(* Logix 5000 project; controller Sucrose_Main Emulate 5570 rev 20.12; software revision 20.01; part 16 of 30 *)
(* tags used below, declared in another part *)
   Alarm_ACK_Master_Timer : TIMER;
   DO_E22_4 : ALIAS FOR FLX_E22:4:O;   // Discrete Output EN2T_FLX 192.168.1.22
   DO_E22_5 : ALIAS FOR FLX_E22:5:O;   // Discrete Output EN2T_FLX 192.168.1.22
   FV230502_AOI : QSI_Flow_Valve;   // FV-23-05-02 PRE FILTER TRAIN 1 INLET LOW POINT DRAIN VALVE
   FV230503_AOI : QSI_Flow_Valve;   // FV-23-05-03 PRE FILTER TRAIN 1 INLET LOW POINT DRAIN VALVE
   FV230504_AOI : QSI_Flow_Valve;   // FV-23-05-04 PRE FILTER TRAIN 1 OUTLET LOW POINT DRAIN VALVE
   FV230505_AOI : QSI_Flow_Valve;   // FV-23-05-05 PRE FILTER TRAIN 1 OUTLET LOW POINT DRAIN VALVE
   FV230509_AOI : QSI_Flow_Valve;   // FV-23-05-09 FINAL FILTER TRAIN 1 INLET LOW POINT DRAIN VALVE
   FV230510_AOI : QSI_Flow_Valve;   // FV-23-05-10 FINAL FILTER TRAIN 1 INLET LOW POINT DRAIN VALVE
   FV230511_AOI : QSI_Flow_Valve;   // FV-23-05-11 FINAL FILTER TRAIN 1 OUTLET LOW POINT DRAIN VALVE
   FV230512_AOI : QSI_Flow_Valve;   // FV-23-05-12 FINAL FILTER TRAIN 1 OUTLET LOW POINT DRAIN VALVE
   Sucrose_MM_Enable : BOOL;
   SucroseCIP_FILTRATION_REMOTE : CIP_REMOTE;
   SucroseFiltration : Area_Program;
(* FiltrationArea_EN2T_IO_Discrete_DO_E22_4, continued *)

ROUTINE _07_FV230502   (* ladder *)
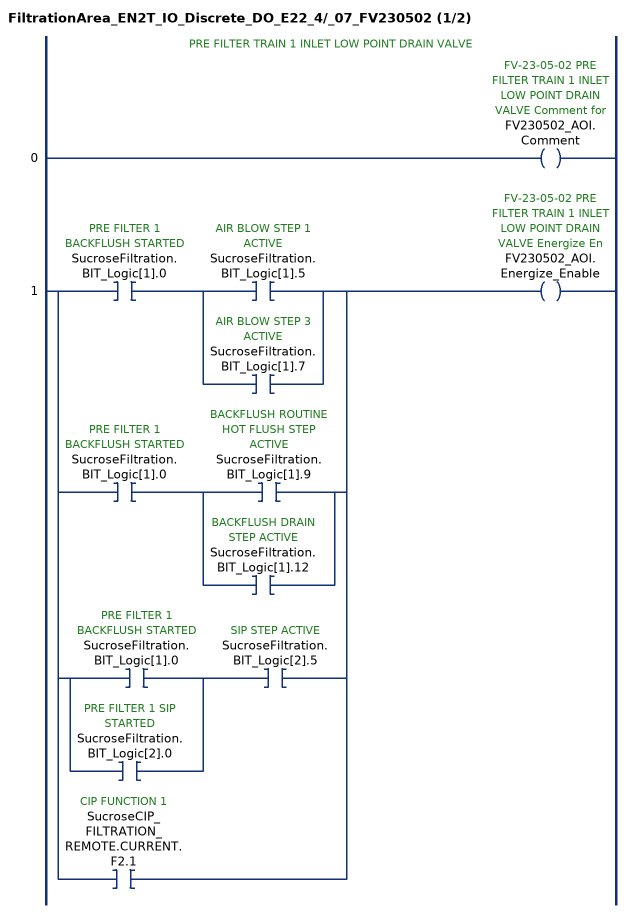
   // PRE FILTER TRAIN 1 INLET LOW POINT DRAIN VALVE
   0: OTE(FV230502_AOI.Comment);
   1: [XIC(SucroseFiltration.BIT_Logic[1].0) [XIC(SucroseFiltration.BIT_Logic[1].5) ,XIC(SucroseFiltration.BIT_Logic[1].7) ] ,XIC(SucroseFiltration.BIT_Logic[1].0) [XIC(SucroseFiltration.BIT_Logic[1].9) ,XIC(SucroseFiltration.BIT_Logic[1].12) ] ,[XIC(SucroseFiltration.BIT_Logic[1].0) ,XIC(SucroseFiltration.BIT_Logic[2].0) ] XIC(SucroseFiltration.BIT_Logic[2].5) ,XIC(SucroseCIP_FILTRATION_REMOTE.CURRENT.F2.1) ]OTE(FV230502_AOI.Energize_Enable);
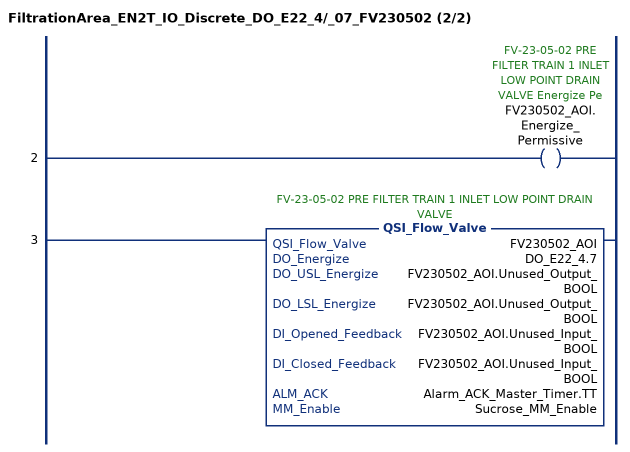
   2: OTE(FV230502_AOI.Energize_Permissive);
   3: QSI_Flow_Valve(FV230502_AOI,DO_E22_4.7,FV230502_AOI.Unused_Output_BOOL,FV230502_AOI.Unused_Output_BOOL,FV230502_AOI.Unused_Input_BOOL,FV230502_AOI.Unused_Input_BOOL,Alarm_ACK_Master_Timer.TT,Sucrose_MM_Enable);
END_ROUTINE

ROUTINE _08_FV230503   (* ladder *)
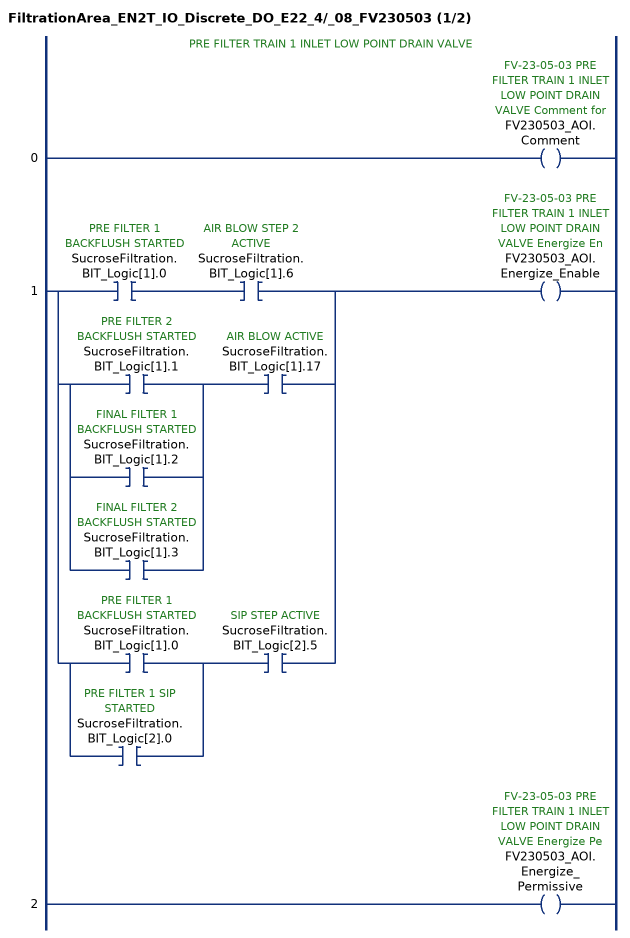
   // PRE FILTER TRAIN 1 INLET LOW POINT DRAIN VALVE
   0: OTE(FV230503_AOI.Comment);
   1: [XIC(SucroseFiltration.BIT_Logic[1].0) XIC(SucroseFiltration.BIT_Logic[1].6) ,[XIC(SucroseFiltration.BIT_Logic[1].1) ,XIC(SucroseFiltration.BIT_Logic[1].2) ,XIC(SucroseFiltration.BIT_Logic[1].3) ] XIC(SucroseFiltration.BIT_Logic[1].17) ,[XIC(SucroseFiltration.BIT_Logic[1].0) ,XIC(SucroseFiltration.BIT_Logic[2].0) ] XIC(SucroseFiltration.BIT_Logic[2].5) ]OTE(FV230503_AOI.Energize_Enable);
   2: OTE(FV230503_AOI.Energize_Permissive);
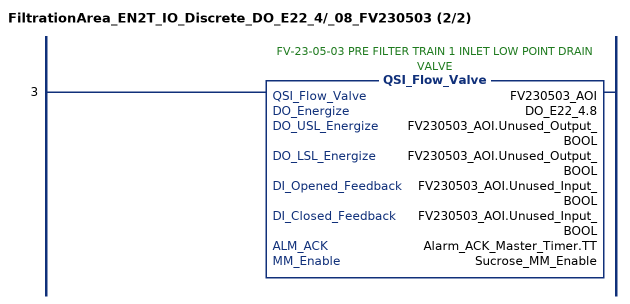
   3: QSI_Flow_Valve(FV230503_AOI,DO_E22_4.8,FV230503_AOI.Unused_Output_BOOL,FV230503_AOI.Unused_Output_BOOL,FV230503_AOI.Unused_Input_BOOL,FV230503_AOI.Unused_Input_BOOL,Alarm_ACK_Master_Timer.TT,Sucrose_MM_Enable);
END_ROUTINE

ROUTINE _09_FV230504   (* ladder *)
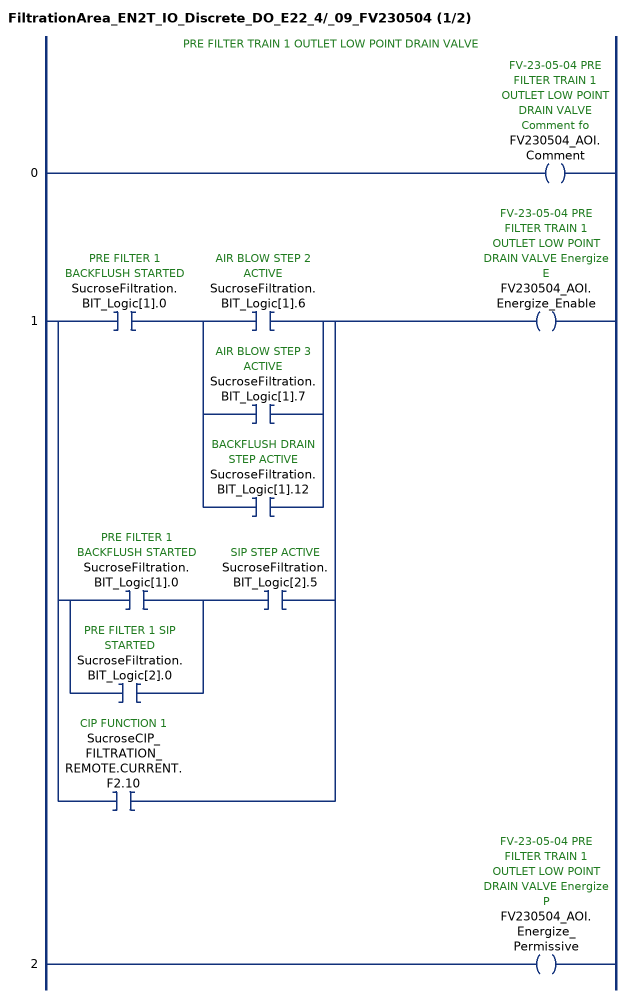
   // PRE FILTER TRAIN 1 OUTLET LOW POINT DRAIN VALVE
   0: OTE(FV230504_AOI.Comment);
   1: [XIC(SucroseFiltration.BIT_Logic[1].0) [XIC(SucroseFiltration.BIT_Logic[1].6) ,XIC(SucroseFiltration.BIT_Logic[1].7) ,XIC(SucroseFiltration.BIT_Logic[1].12) ] ,[XIC(SucroseFiltration.BIT_Logic[1].0) ,XIC(SucroseFiltration.BIT_Logic[2].0) ] XIC(SucroseFiltration.BIT_Logic[2].5) ,XIC(SucroseCIP_FILTRATION_REMOTE.CURRENT.F2.10) ]OTE(FV230504_AOI.Energize_Enable);
   2: OTE(FV230504_AOI.Energize_Permissive);
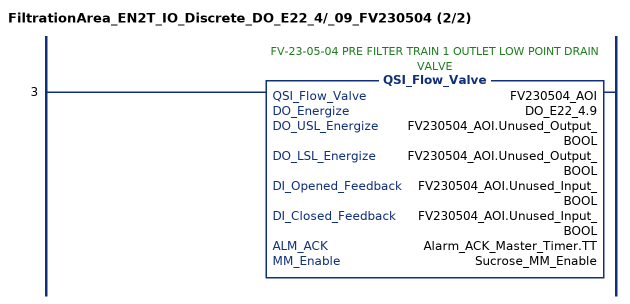
   3: QSI_Flow_Valve(FV230504_AOI,DO_E22_4.9,FV230504_AOI.Unused_Output_BOOL,FV230504_AOI.Unused_Output_BOOL,FV230504_AOI.Unused_Input_BOOL,FV230504_AOI.Unused_Input_BOOL,Alarm_ACK_Master_Timer.TT,Sucrose_MM_Enable);
END_ROUTINE

ROUTINE _10_FV230505   (* ladder *)
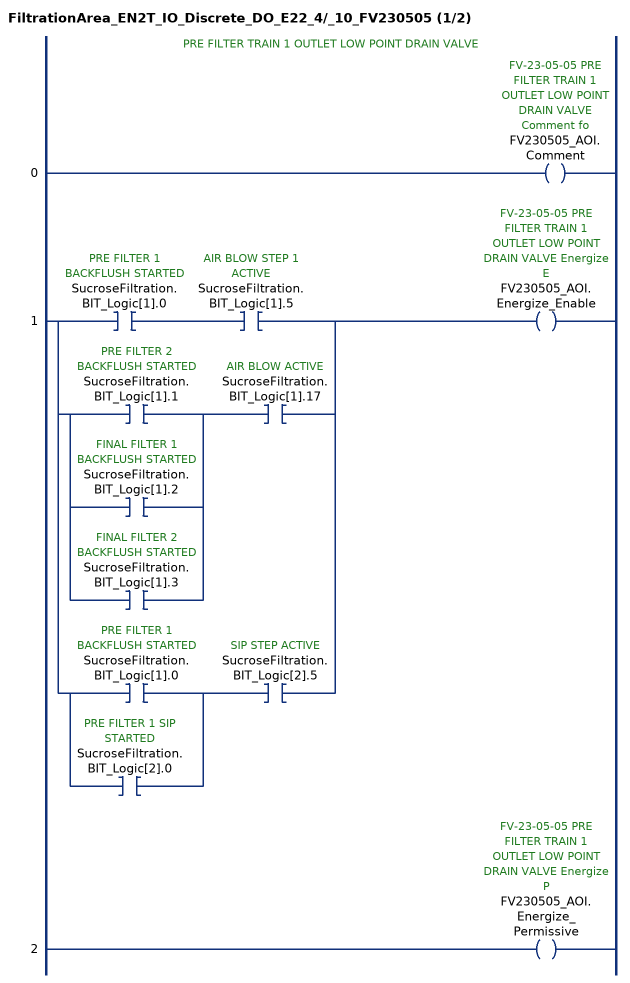
   // PRE FILTER TRAIN 1 OUTLET LOW POINT DRAIN VALVE
   0: OTE(FV230505_AOI.Comment);
   1: [XIC(SucroseFiltration.BIT_Logic[1].0) XIC(SucroseFiltration.BIT_Logic[1].5) ,[XIC(SucroseFiltration.BIT_Logic[1].1) ,XIC(SucroseFiltration.BIT_Logic[1].2) ,XIC(SucroseFiltration.BIT_Logic[1].3) ] XIC(SucroseFiltration.BIT_Logic[1].17) ,[XIC(SucroseFiltration.BIT_Logic[1].0) ,XIC(SucroseFiltration.BIT_Logic[2].0) ] XIC(SucroseFiltration.BIT_Logic[2].5) ]OTE(FV230505_AOI.Energize_Enable);
   2: OTE(FV230505_AOI.Energize_Permissive);
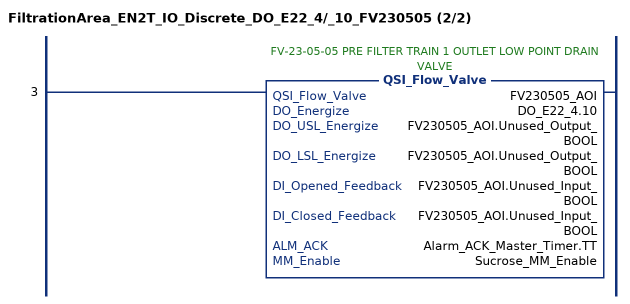
   3: QSI_Flow_Valve(FV230505_AOI,DO_E22_4.10,FV230505_AOI.Unused_Output_BOOL,FV230505_AOI.Unused_Output_BOOL,FV230505_AOI.Unused_Input_BOOL,FV230505_AOI.Unused_Input_BOOL,Alarm_ACK_Master_Timer.TT,Sucrose_MM_Enable);
END_ROUTINE

ROUTINE _11_FV230509   (* ladder *)
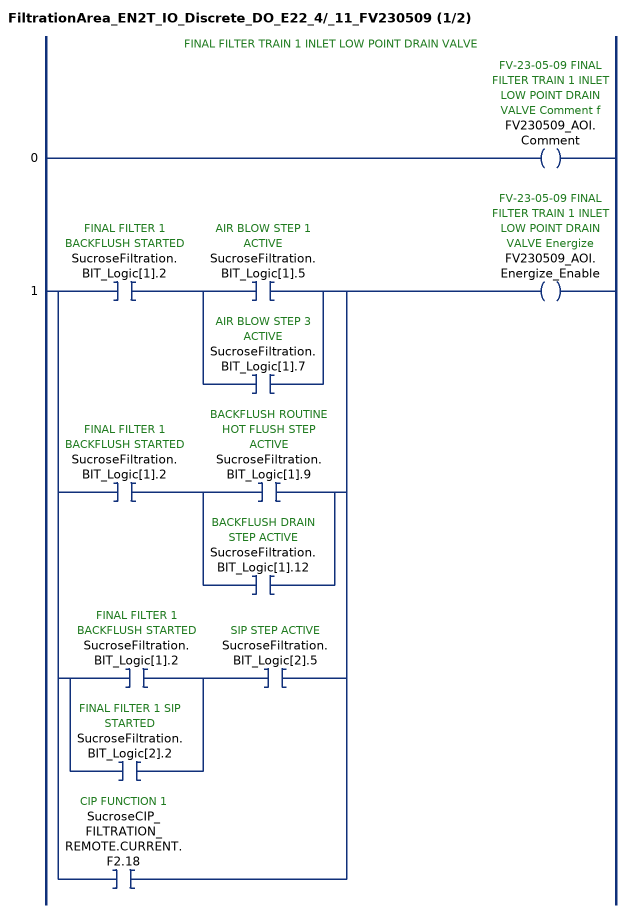
   // FINAL FILTER TRAIN 1 INLET LOW POINT DRAIN VALVE
   0: OTE(FV230509_AOI.Comment);
   1: [XIC(SucroseFiltration.BIT_Logic[1].2) [XIC(SucroseFiltration.BIT_Logic[1].5) ,XIC(SucroseFiltration.BIT_Logic[1].7) ] ,XIC(SucroseFiltration.BIT_Logic[1].2) [XIC(SucroseFiltration.BIT_Logic[1].9) ,XIC(SucroseFiltration.BIT_Logic[1].12) ] ,[XIC(SucroseFiltration.BIT_Logic[1].2) ,XIC(SucroseFiltration.BIT_Logic[2].2) ] XIC(SucroseFiltration.BIT_Logic[2].5) ,XIC(SucroseCIP_FILTRATION_REMOTE.CURRENT.F2.18) ]OTE(FV230509_AOI.Energize_Enable);
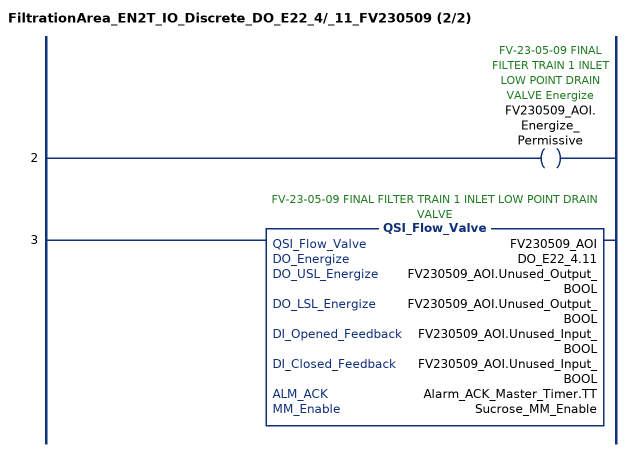
   2: OTE(FV230509_AOI.Energize_Permissive);
   3: QSI_Flow_Valve(FV230509_AOI,DO_E22_4.11,FV230509_AOI.Unused_Output_BOOL,FV230509_AOI.Unused_Output_BOOL,FV230509_AOI.Unused_Input_BOOL,FV230509_AOI.Unused_Input_BOOL,Alarm_ACK_Master_Timer.TT,Sucrose_MM_Enable);
END_ROUTINE

ROUTINE MainRoutine   (* ladder *)
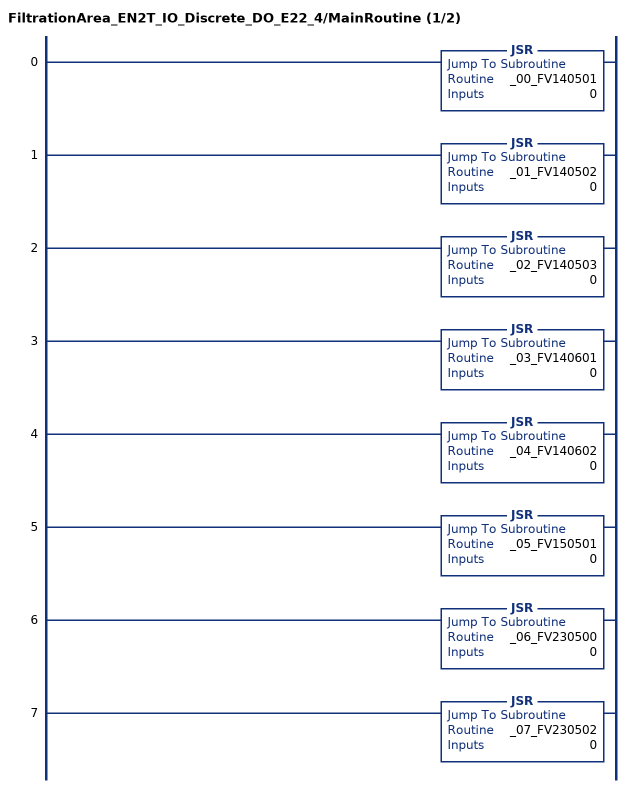
   0: JSR(_00_FV140501,0);
   1: JSR(_01_FV140502,0);
   2: JSR(_02_FV140503,0);
   3: JSR(_03_FV140601,0);
   4: JSR(_04_FV140602,0);
   5: JSR(_05_FV150501,0);
   6: JSR(_06_FV230500,0);
   7: JSR(_07_FV230502,0);
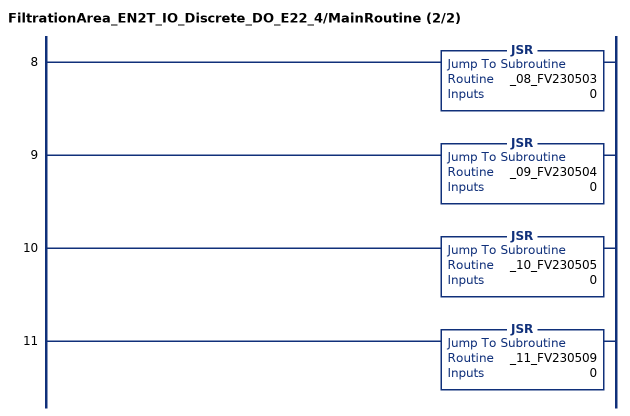
   8: JSR(_08_FV230503,0);
   9: JSR(_09_FV230504,0);
   10: JSR(_10_FV230505,0);
   11: JSR(_11_FV230509,0);
END_ROUTINE
END_PROGRAM

PROGRAM FiltrationArea_EN2T_IO_Discrete_DO_E22_5   (* main routine MainRoutine *)

ROUTINE _00_FV230510   (* ladder *)
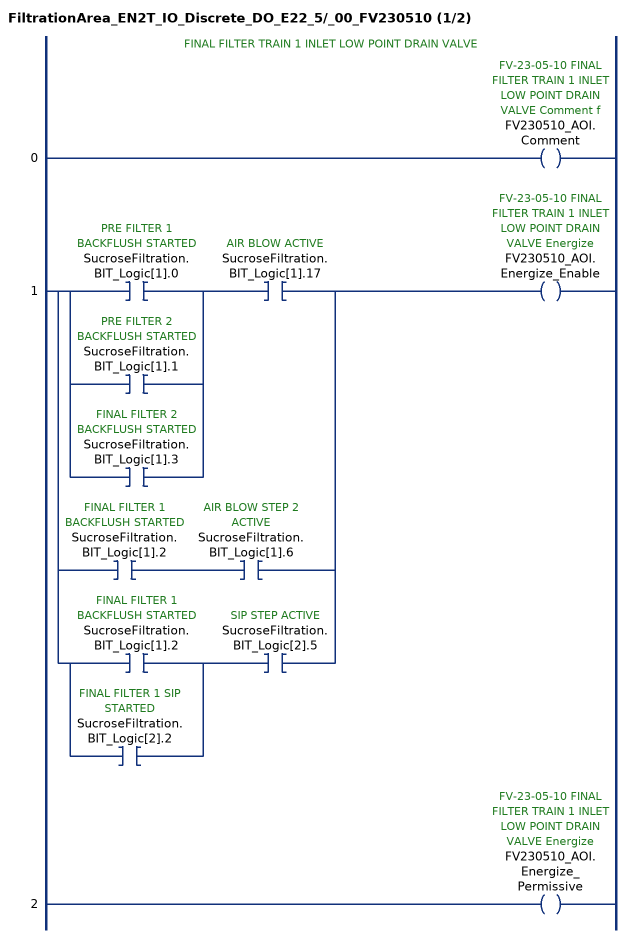
   // FINAL FILTER TRAIN 1 INLET LOW POINT DRAIN VALVE
   0: OTE(FV230510_AOI.Comment);
   1: [[XIC(SucroseFiltration.BIT_Logic[1].0) ,XIC(SucroseFiltration.BIT_Logic[1].1) ,XIC(SucroseFiltration.BIT_Logic[1].3) ] XIC(SucroseFiltration.BIT_Logic[1].17) ,XIC(SucroseFiltration.BIT_Logic[1].2) XIC(SucroseFiltration.BIT_Logic[1].6) ,[XIC(SucroseFiltration.BIT_Logic[1].2) ,XIC(SucroseFiltration.BIT_Logic[2].2) ] XIC(SucroseFiltration.BIT_Logic[2].5) ]OTE(FV230510_AOI.Energize_Enable);
   2: OTE(FV230510_AOI.Energize_Permissive);
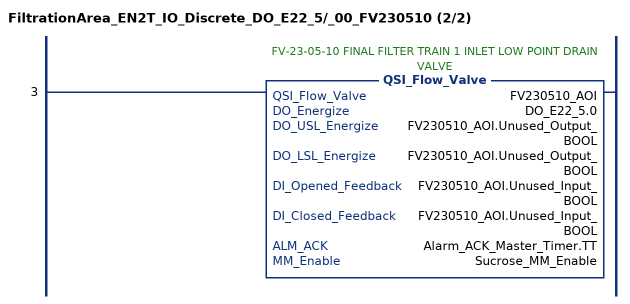
   3: QSI_Flow_Valve(FV230510_AOI,DO_E22_5.0,FV230510_AOI.Unused_Output_BOOL,FV230510_AOI.Unused_Output_BOOL,FV230510_AOI.Unused_Input_BOOL,FV230510_AOI.Unused_Input_BOOL,Alarm_ACK_Master_Timer.TT,Sucrose_MM_Enable);
END_ROUTINE

ROUTINE _01_FV230511   (* ladder *)
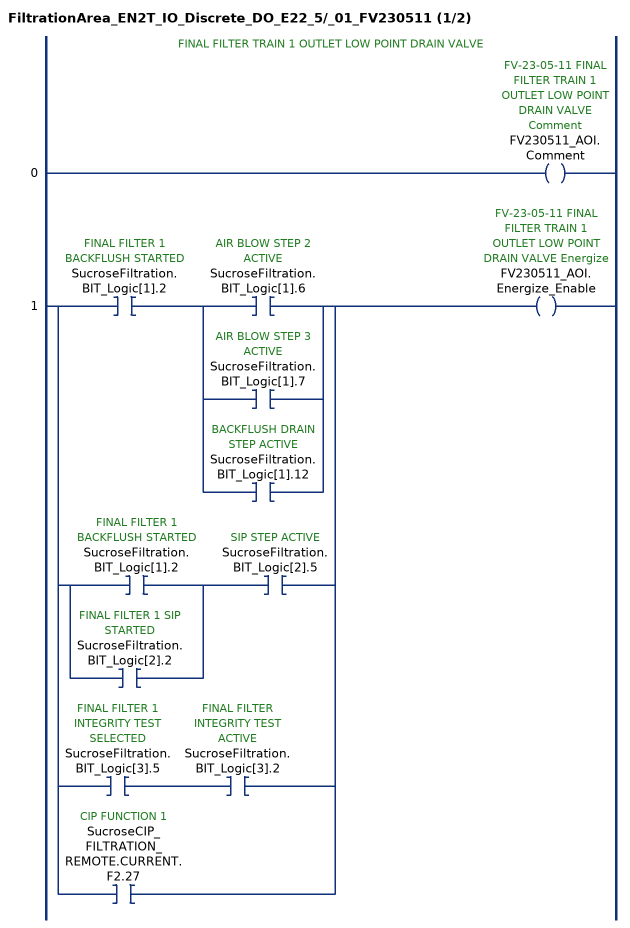
   // FINAL FILTER TRAIN 1 OUTLET LOW POINT DRAIN VALVE
   0: OTE(FV230511_AOI.Comment);
   1: [XIC(SucroseFiltration.BIT_Logic[1].2) [XIC(SucroseFiltration.BIT_Logic[1].6) ,XIC(SucroseFiltration.BIT_Logic[1].7) ,XIC(SucroseFiltration.BIT_Logic[1].12) ] ,[XIC(SucroseFiltration.BIT_Logic[1].2) ,XIC(SucroseFiltration.BIT_Logic[2].2) ] XIC(SucroseFiltration.BIT_Logic[2].5) ,XIC(SucroseFiltration.BIT_Logic[3].5) XIC(SucroseFiltration.BIT_Logic[3].2) ,XIC(SucroseCIP_FILTRATION_REMOTE.CURRENT.F2.27) ]OTE(FV230511_AOI.Energize_Enable);
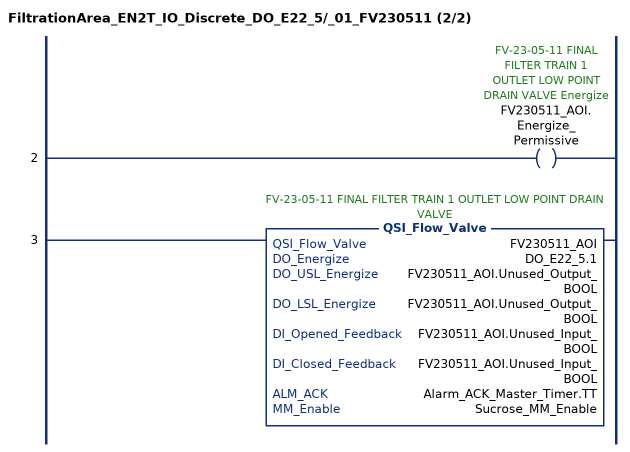
   2: OTE(FV230511_AOI.Energize_Permissive);
   3: QSI_Flow_Valve(FV230511_AOI,DO_E22_5.1,FV230511_AOI.Unused_Output_BOOL,FV230511_AOI.Unused_Output_BOOL,FV230511_AOI.Unused_Input_BOOL,FV230511_AOI.Unused_Input_BOOL,Alarm_ACK_Master_Timer.TT,Sucrose_MM_Enable);
END_ROUTINE

ROUTINE _02_FV230512   (* ladder *)
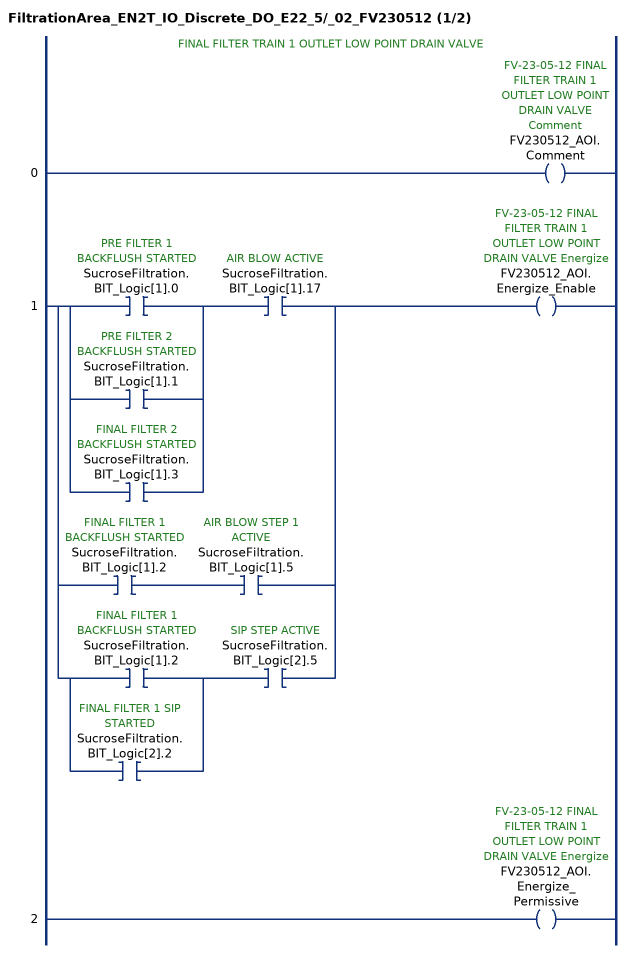
   // FINAL FILTER TRAIN 1 OUTLET LOW POINT DRAIN VALVE
   0: OTE(FV230512_AOI.Comment);
   1: [[XIC(SucroseFiltration.BIT_Logic[1].0) ,XIC(SucroseFiltration.BIT_Logic[1].1) ,XIC(SucroseFiltration.BIT_Logic[1].3) ] XIC(SucroseFiltration.BIT_Logic[1].17) ,XIC(SucroseFiltration.BIT_Logic[1].2) XIC(SucroseFiltration.BIT_Logic[1].5) ,[XIC(SucroseFiltration.BIT_Logic[1].2) ,XIC(SucroseFiltration.BIT_Logic[2].2) ] XIC(SucroseFiltration.BIT_Logic[2].5) ]OTE(FV230512_AOI.Energize_Enable);
   2: OTE(FV230512_AOI.Energize_Permissive);
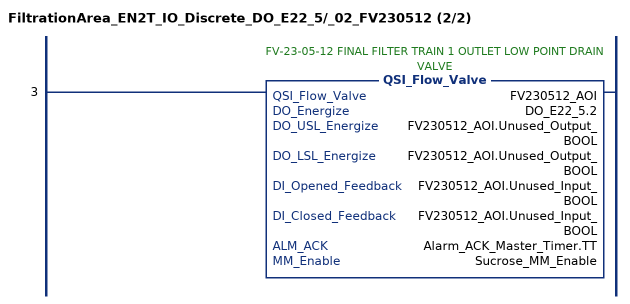
   3: QSI_Flow_Valve(FV230512_AOI,DO_E22_5.2,FV230512_AOI.Unused_Output_BOOL,FV230512_AOI.Unused_Output_BOOL,FV230512_AOI.Unused_Input_BOOL,FV230512_AOI.Unused_Input_BOOL,Alarm_ACK_Master_Timer.TT,Sucrose_MM_Enable);
END_ROUTINE
